INTERFACE I_UserDefinedDatatype EXTENDS I_Datatype

PROPERTY PUBLIC Identifier : T_MAXSTRING
GET
END_GET
END_PROPERTY

END_INTERFACE

(* stored: Version 1.1.0.1, ProductVersion 3.1.4024.12
   Itf I_UserDefinedDatatype: Id {60aa8cd6-0b23-0d67-0233-1aa454e3e8a0}
   Property Identifier: Id {c0b81c95-7f74-08ff-33a3-1876d9b8949f}
   Get Get: Id {c077c9be-21ce-0f58-3320-fceb8f1fd1a7} *)
